(* Logix 5000 project; controller Ceca_1650T_Press 5069-L306ERM rev 32.11; software revision 32.02 *)

TASK MainTask (continuous, watchdog 500 ms) : MainProgram

MODULES
   Local : 5069-L306ERM (5069 0, rev 32.11)
      INPUT2 : vendor 1 type 7 code 1212 (5069 2, rev 3.1, StandardDataDriven RPI 5 ms)
      INPUT3 : vendor 1 type 7 code 1212 (5069 3, rev 3.1, StandardDataDriven RPI 5 ms)
      INPUT1 : vendor 1 type 7 code 1212 (5069 1, rev 3.1, StandardDataDriven RPI 5 ms)
      OUTPUT1 : vendor 1 type 7 code 1215 (5069 4, rev 3.1, StandardDataDriven RPI 5 ms)
      OUTPUT3 : vendor 1 type 7 code 1215 (5069 6, rev 3.1, StandardDataDriven RPI 5 ms)
      OUTPUT2 : vendor 1 type 7 code 1215 (5069 5, rev 3.1, StandardDataDriven RPI 5 ms)
END_MODULES

VAR_GLOBAL   (* controller tags *)
   AIR_SUPPLY_PRESSURE_DETECT : BOOL;
   AUTO_CYCLE_ENABLED : BOOL;   // M0014 HMI SELECTION
   AUTO_CYCLE_SELECTED : BOOL;   // HMI BUTTON/SELECTION B0102
   AUTO_CYCLE_STOP_PB : BOOL;
   AUTO_LOWER_LIMIT : BOOL;   // ENCODER SIGNAL B0155
   AUTO_ONE_CYCLE_ENABLED : BOOL;   // M0013 HMI SELECTION
   AUTO_ONE_CYCLE_SELECTED : BOOL;   // HMI BUTTON/SELECTION B0101
   AUTO_RESET_ALLOWED : BOOL;   // M003E
   AUTO_START_PB : BOOL;
   AUTO_START_PB_RESET : BOOL;
   AUTO_UPPER_LIMIT : BOOL;   // ENCODER SIGNAL B0151
   BLANKING_OFF_SIGNAL : TIMER := (PRE := 150);   // T0018
   BLANKING_PS_ENABLED : BOOL;   // M0018
   BOLSTER_CLAMP_OFF_LIMIT : BOOL;   // B0013
   BOLSTER_CLAMP_OFF_VALVE : BOOL;
   BOLSTER_CLAMP_ON : BOOL;   // M0006
   BOLSTER_CLAMP_ON_LIMIT : BOOL;   // B0012
   BOLSTER_CLAMP_ON_VALVE : BOOL;
   BOLSTER_DISABLED : BOOL;   // M0010
   BOLSTER_IN_ASSIST_LIMIT : BOOL;
   BOLSTER_IN_LIMIT : BOOL;   // B000E
   BOLSTER_IN_VALVE : BOOL;
   BOLSTER_LIFT_PRESSURE_DETECT : BOOL;
   BOLSTER_OUT_ASSIST_LIMIT : BOOL;
   BOLSTER_OUT_LIMIT : BOOL;
   BOLSTER_OUT_VALVE : BOOL;
   BOLSTER_REDUCTION_VALVE : BOOL;
   BOLSTER_TOUCH_LIMIT_1 : BOOL;   // B0014
   BOLSTER_TOUCH_LIMIT_2 : BOOL;   // B0015
   BOTH_DIE_CUSHIONS_DOWN : BOOL;   // M0036
   BUZZER_SIGNAL : BOOL;
   CANCEL_CYLINDER_LOWER_LIMIT : BOOL;
   CANCEL_DECOMPRESSION_VALVE : BOOL;
   CANCEL_HIGH_PRESSURE_VAVLE : BOOL;
   CANCEL_LOW_PRESSURE_VALVE : BOOL;
   CANCEL_UP_VALVE : BOOL;
   COOLING_WATER_ON_VALVE : BOOL;
   DC_POWER_ASSIST_VALVE : BOOL;
   DEBOUNCE_TIMER_LOCKING_OFF : TIMER := (PRE := 100);
   DEBOUNCE_TIMER_LOCKING_OFF_COMPLETE : TIMER := (PRE := 100);
   DECOMPRESSION : BOOL;   // M006D
   DIE_CHANGE_ENABLED : BOOL;   // M0015
   DIE_CHANGE_MODE : BOOL;   // HMI BUTTON/SELECTION B0103
   DIE_CUSHION_PB_OFF_STATE : BOOL;   // M003F
   DIE_DRAWRIC_CYLINDER_UPPER_PS : BOOL;   // B0018
   DIE_DRAWRIC_DECOMPRESSION_VALVE : BOOL;
   DIE_DRAWRIC_POWER_ASSIST_VALVE : BOOL;
   DIE_SET_CHANGING : BOOL;
   DIECUSHION_PUMP_UNLOADING_VALVE_1 : BOOL;
   DIECUSHION_PUMP_UNLOADING_VALVE_2 : BOOL;
   DIECUSHION_UPPER_LIMIT : BOOL;
   DRAW_ASSIST_COMPLETE : BOOL;   // M007D
   DRAW_BLANKING_NOT_SELECT : BOOL;   // M0017
   DRAW_UP_ASSIST : BOOL;   // M007C
   DRAWING_LS_ENABLED : BOOL;   // M0016????REMOVE????
   EMERGENCY_STOP : BOOL;
   ENABLE_1000T : BOOL;   // HMI BUTTON/RECIPE
   ENABLE_1500T : BOOL;   // HMI BUTTON/RECIPE
   ENABLE_500T : BOOL;   // HMI BUTTON/RECIPE
   FILTER_CHOKER : BOOL;
   FRONT_SHUTTER_SAFETY : BOOL;   // M002A
   FRONT_SUTTER_ON_LIMIT : BOOL;
   HALF_FINISHED_CYLINDER_ADVANCE_LIMIT : BOOL;
   HALF_FINISHED_CYLINDER_RETURN_LIMIT : BOOL;
   HALF_FINISHED_SUPPLY_VALVE : BOOL;
   INCH_ENABLED : BOOL;   // M0012 HMI SELECTION
   INCHING_SELECTED : BOOL;   // HMI BUTTON/SELECTION B0100
   L_DIECUSHION_AUTO_UP_LIMIT : BOOL;   // B0156 ENCODER SIGNAL
   L_DIECUSHION_DOWN : BOOL;   // M0003
   L_DIECUSHION_UP : BOOL;   // M0002
   LEFT_DIECUSHION_DECOMPRESSION_VALVE : BOOL;
   LEFT_DIECUSHION_DOWN_VALVE : BOOL;
   LEFT_DIECUSHION_LOWER_LIMIT : BOOL;   // B0006
   LEFT_DIECUSHION_POWER_ASSIST_VALVE : BOOL;
   LEFT_DIECUSHION_UP_VALVE : BOOL;
   LEFT_DIECUSHION_UPPER_LIMIT : BOOL;   // B0005
   LIFT_CYLINDER_DOWN_VALVE : BOOL;
   LIFT_CYLINDER_UP_VALVE : BOOL;
   LOCKING_OFF : BOOL;   // M0004
   LOCKING_OFF_ASSIST : BOOL;   // M0032
   LOCKING_OFF_COMPLETE : BOOL;   // M0033
   LOCKING_OFF_LIMIT : BOOL;   // B0007
   LOCKING_OFF_MEMORY : BOOL;   // M0031
   LOCKING_OFF_VALVE : BOOL;   // B0058
   LOCKING_ON : BOOL;   // M0005
   LOCKING_ON_LIMIT : BOOL;   // B0008
   LUBRICATION_OIL_LEVEL_DETECT : BOOL;
   LUBRICATION_PRESSURE_DETECT : BOOL;
   M_PRESS_DOWN : BOOL;   // M006A
   M_PRESS_DOWN_COMPLETE : BOOL;   // M006C
   M_PRESS_DOWN_COMPLETE_TIMER : TIMER := (PRE := 30);   // T0012
   M_PRESS_UP : BOOL;   // M006E
   M_PRESS_UP_COMPLETE : BOOL;   // M006F
   MAIN_DOWN_VALVE : BOOL;   // B0041
   MAIN_DOWN_VALVE_1000_TON : BOOL;   // B0043
   MAIN_DOWN_VALVE_500_TON : BOOL;   // B0042
   MAIN_LOWER_ASSIST_LIMIT : BOOL;   // B0026
   MAIN_LOWER_LIMIT : BOOL;   // B0002
   MAIN_NO_LOAD_VALVE : BOOL;   // B0046
   MAIN_POWER_HOLDING_VALVE : BOOL;   // B0045
   MAIN_PRESS_CONDITION_DOWN : BOOL;   // M0039
   MAIN_PRESS_CONDITION_UP : BOOL;   // M0038
   MAIN_PRESS_DOWN : BOOL;   // M0045
   MAIN_PRESS_DOWN_ASSIST : BOOL;   // M0044
   MAIN_PRESS_DOWN_MEMORY : BOOL;   // M006A
   MAIN_PRESS_NO_PRESSURE_DOWN : BOOL;   // M0047
   MAIN_PRESS_PRESSURE_DETECT : BOOL;   // B0016
   MAIN_PRESS_SLOW_DOWN : BOOL;   // M0046
   MAIN_PRESS_SLOW_DOWN_SIGNAL : BOOL;   // M0030
   MAIN_PRESS_SLOW_UP : BOOL;   // M0042
   MAIN_PRESS_UP : BOOL;   // M0041
   MAIN_PRESS_UP_ASSIST : BOOL;   // M0040
   MAIN_SLOW_DOWN_VALVE : BOOL;   // B0044
   MAIN_UP_VALVE : BOOL;   // B0040
   MAIN_UPPER_ASSIST : BOOL;   // B0001
   MAIN_UPPER_LIMIT : BOOL;   // B0000
   MOTOR_OVER_LOAD : BOOL;
   NO_PRESSUE_DOWN_PB : BOOL;   // B010D HMI BUTTON
   OIL_COOLER_START : BOOL;
   OIL_TEMP_TOO_HIGH : BOOL;
   OIL_TEMP_WARM_UP_START : BOOL;
   OPERATION_ON : BOOL;   // B0020
   PILOT_CHECK_OPEN_VALVE : BOOL;   // B0048
   PILOT_PUMP_HIGH_PRESSURE_VALVE : BOOL;
   PILOT_PUMP_MIDDLE_PRESSURE_VALVE : BOOL;
   PILOT_PUMP_ON : BOOL;
   PREFILL_VALVE_OPEN_VALVE : BOOL;   // B0047
   PREFILL_VALVE_OPEN_VALVE_2 : BOOL;
   PRESS_AUTO_CYCLE_SELECT_CONDITION : BOOL;   // M0060
   PRESS_AUTO_RUN : BOOL;   // M0069
   PRESS_HAS_A_FAULT_2 : BOOL;   // M0028
   PRESS_HOLDING_TIME : BOOL;   // M006B
   PRESS_HOLDING_TIMER : TIMER;   // PRESS HOLDING TIMER
   PRESS_READY_CONFIRM : BOOL;   // M0043
   PUMP_RUN : BOOL;   // B0021
   PUMP_STOP_SIGNAL : BOOL;
   R_DIECUSHION_AUTO_UP_LIMIT : BOOL;   // B0158 ENCODER SIGNAL
   R_DIECUSHION_DOWN : BOOL;   // M0001
   R_DIECUSHION_UP : BOOL;   // M0000
   REAR_SHUTTER_ON_LIMIT : BOOL;
   RIGHT_DIECUSHION_DECOMPRESSION_VALVE : BOOL;
   RIGHT_DIECUSHION_DOWN_VALVE : BOOL;
   RIGHT_DIECUSHION_LOWER_LIMIT : BOOL;   // B0004
   RIGHT_DIECUSHION_POWER_ASSIST_VALVE : BOOL;
   RIGHT_DIECUSHION_UP_VALVE : BOOL;
   RIGHT_DIECUSHION_UPPER_LIMIT : BOOL;   // B0003
   SAFETY_BAR_OPENED : BOOL;   // B000B
   SLIDE_DOWN_PB : BOOL;   // B010B HMI BUTTON
   SLIDE_SLOW_DOWN_PB : BOOL;   // B010C HMI BUTTON
   SLIDE_SLOW_DOWN_SIGNAL : BOOL;   // B0154 ENCODER SIGNAL
   SLIDE_SLOW_UP_PB : BOOL;   // B010A HMI BUTTON
   SLIDE_UP_PB : BOOL;   // HMI BUTTON B0109
   TIMER_OFF_DELAY_1500T : TIMER := (PRE := 50);   // T0017
   TIMER_OFF_DELAY_500T : TIMER := (PRE := 10);   // T0016
   UPPER_DIE_CLAMP_ON_DETECT : BOOL;
   UPPER_DIECLAMP_OFF_VALVE : BOOL;
   WARM_UP_OFF_TEMP : BOOL;
   WORK_LOCATION_VALVE : BOOL;
   WORKING_OIL_LEVEL_DETECT : BOOL;
END_VAR

PROGRAM MainProgram   (* main routine MainRoutine *)
VAR
   MESSAGES : STRING[100];
END_VAR

ROUTINE Bolster   (* ladder *)
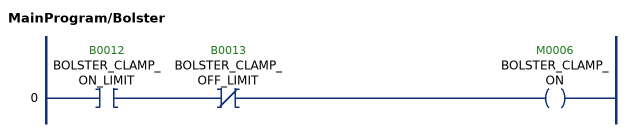
   0: XIC(BOLSTER_CLAMP_ON_LIMIT)XIO(BOLSTER_CLAMP_OFF_LIMIT)OTE(BOLSTER_CLAMP_ON);
END_ROUTINE

ROUTINE Cancel_Valves   (* ladder *)
END_ROUTINE

ROUTINE Die_Cushion   (* ladder *)
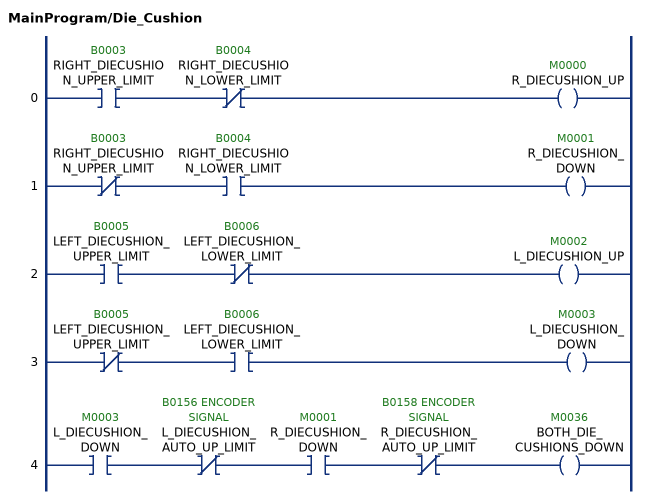
   0: XIC(RIGHT_DIECUSHION_UPPER_LIMIT)XIO(RIGHT_DIECUSHION_LOWER_LIMIT)OTE(R_DIECUSHION_UP);
   1: XIO(RIGHT_DIECUSHION_UPPER_LIMIT)XIC(RIGHT_DIECUSHION_LOWER_LIMIT)OTE(R_DIECUSHION_DOWN);
   2: XIC(LEFT_DIECUSHION_UPPER_LIMIT)XIO(LEFT_DIECUSHION_LOWER_LIMIT)OTE(L_DIECUSHION_UP);
   3: XIO(LEFT_DIECUSHION_UPPER_LIMIT)XIC(LEFT_DIECUSHION_LOWER_LIMIT)OTE(L_DIECUSHION_DOWN);
   4: XIC(L_DIECUSHION_DOWN)XIO(L_DIECUSHION_AUTO_UP_LIMIT)XIC(R_DIECUSHION_DOWN)XIO(R_DIECUSHION_AUTO_UP_LIMIT)OTE(BOTH_DIE_CUSHIONS_DOWN);
END_ROUTINE

ROUTINE Draw   (* ladder *)
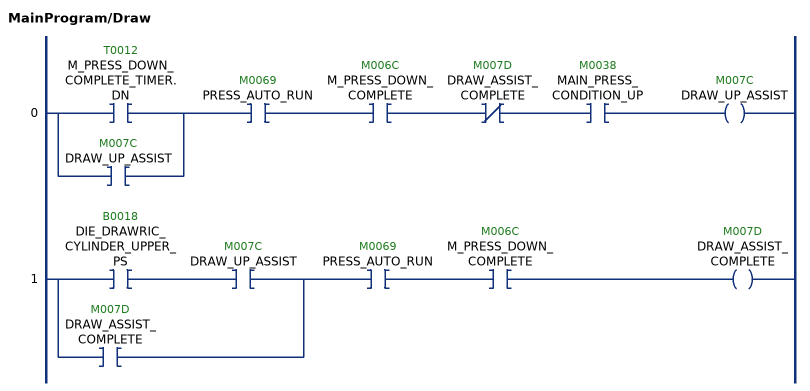
   0: [XIC(M_PRESS_DOWN_COMPLETE_TIMER.DN) ,XIC(DRAW_UP_ASSIST) ]XIC(PRESS_AUTO_RUN)XIC(M_PRESS_DOWN_COMPLETE)XIO(DRAW_ASSIST_COMPLETE)XIC(MAIN_PRESS_CONDITION_UP)OTE(DRAW_UP_ASSIST);
   1: [XIC(DIE_DRAWRIC_CYLINDER_UPPER_PS) XIC(DRAW_UP_ASSIST) ,XIC(DRAW_ASSIST_COMPLETE) ]XIC(PRESS_AUTO_RUN)XIC(M_PRESS_DOWN_COMPLETE)OTE(DRAW_ASSIST_COMPLETE);
END_ROUTINE

ROUTINE Inputs   (* ladder *)
   0: ;
END_ROUTINE

ROUTINE Locking   (* ladder *)
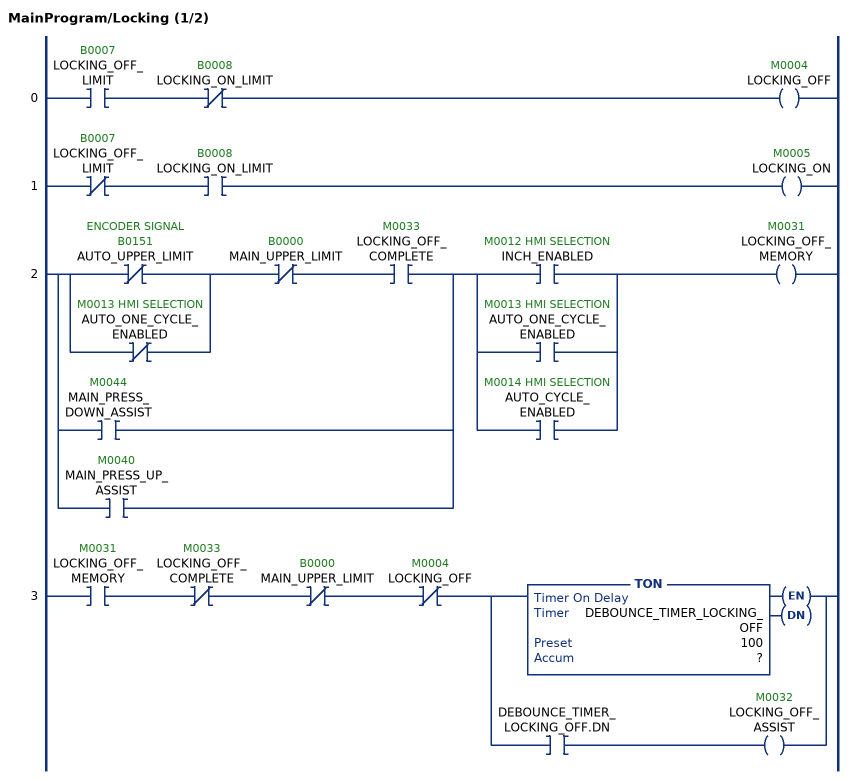
   0: XIC(LOCKING_OFF_LIMIT)XIO(LOCKING_ON_LIMIT)OTE(LOCKING_OFF);
   1: XIO(LOCKING_OFF_LIMIT)XIC(LOCKING_ON_LIMIT)OTE(LOCKING_ON);
   2: [[XIO(AUTO_UPPER_LIMIT) ,XIO(AUTO_ONE_CYCLE_ENABLED) ] XIO(MAIN_UPPER_LIMIT) XIC(LOCKING_OFF_COMPLETE) ,XIC(MAIN_PRESS_DOWN_ASSIST) ,XIC(MAIN_PRESS_UP_ASSIST) ][XIC(INCH_ENABLED) ,XIC(AUTO_ONE_CYCLE_ENABLED) ,XIC(AUTO_CYCLE_ENABLED) ]OTE(LOCKING_OFF_MEMORY);
   3: XIC(LOCKING_OFF_MEMORY)XIO(LOCKING_OFF_COMPLETE)XIO(MAIN_UPPER_LIMIT)XIO(LOCKING_OFF)[TON(DEBOUNCE_TIMER_LOCKING_OFF,?,?) ,XIC(DEBOUNCE_TIMER_LOCKING_OFF.DN) OTE(LOCKING_OFF_ASSIST) ];
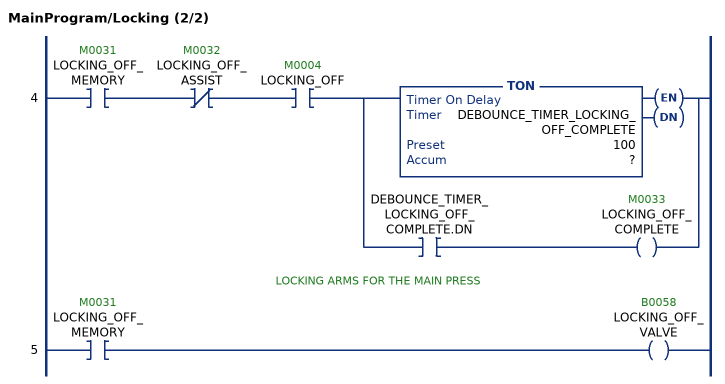
   4: XIC(LOCKING_OFF_MEMORY)XIO(LOCKING_OFF_ASSIST)XIC(LOCKING_OFF)[TON(DEBOUNCE_TIMER_LOCKING_OFF_COMPLETE,?,?) ,XIC(DEBOUNCE_TIMER_LOCKING_OFF_COMPLETE.DN) OTE(LOCKING_OFF_COMPLETE) ];
   // LOCKING ARMS FOR THE MAIN PRESS
   5: XIC(LOCKING_OFF_MEMORY)OTE(LOCKING_OFF_VALVE);
END_ROUTINE

ROUTINE Main_Down   (* ladder *)
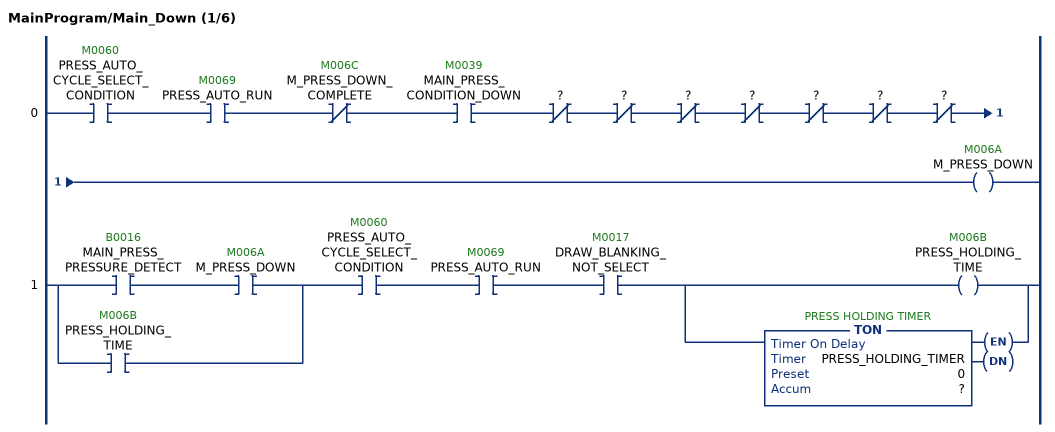
   0: XIC(PRESS_AUTO_CYCLE_SELECT_CONDITION)XIC(PRESS_AUTO_RUN)XIO(M_PRESS_DOWN_COMPLETE)XIC(MAIN_PRESS_CONDITION_DOWN)XIO(?)XIO(?)XIO(?)XIO(?)XIO(?)XIO(?)XIO(?)OTE(M_PRESS_DOWN);
   1: [XIC(MAIN_PRESS_PRESSURE_DETECT) XIC(M_PRESS_DOWN) ,XIC(PRESS_HOLDING_TIME) ]XIC(PRESS_AUTO_CYCLE_SELECT_CONDITION)XIC(PRESS_AUTO_RUN)XIC(DRAW_BLANKING_NOT_SELECT)[OTE(PRESS_HOLDING_TIME) ,TON(PRESS_HOLDING_TIMER,?,?) ];
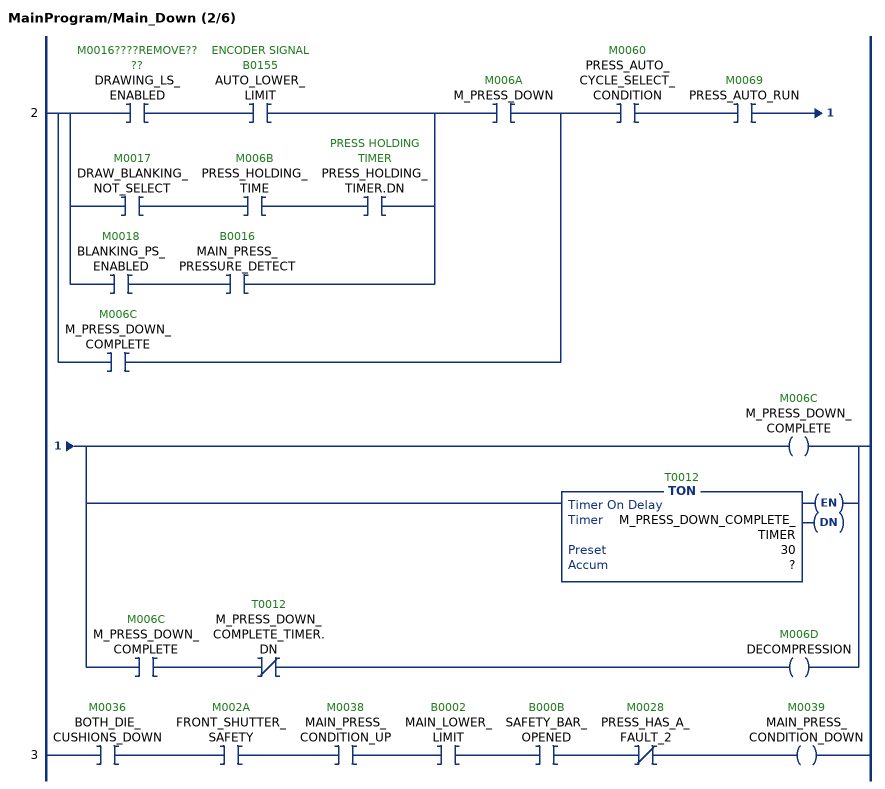
   2: [[XIC(DRAWING_LS_ENABLED) XIC(AUTO_LOWER_LIMIT) ,XIC(DRAW_BLANKING_NOT_SELECT) XIC(PRESS_HOLDING_TIME) XIC(PRESS_HOLDING_TIMER.DN) ,XIC(BLANKING_PS_ENABLED) XIC(MAIN_PRESS_PRESSURE_DETECT) ] XIC(M_PRESS_DOWN) ,XIC(M_PRESS_DOWN_COMPLETE) ]XIC(PRESS_AUTO_CYCLE_SELECT_CONDITION)XIC(PRESS_AUTO_RUN)[OTE(M_PRESS_DOWN_COMPLETE) ,TON(M_PRESS_DOWN_COMPLETE_TIMER,?,?) ,XIC(M_PRESS_DOWN_COMPLETE) XIO(M_PRESS_DOWN_COMPLETE_TIMER.DN) OTE(DECOMPRESSION) ];
   3: XIC(BOTH_DIE_CUSHIONS_DOWN)XIC(FRONT_SHUTTER_SAFETY)XIC(MAIN_PRESS_CONDITION_UP)XIC(MAIN_LOWER_LIMIT)XIC(SAFETY_BAR_OPENED)XIO(PRESS_HAS_A_FAULT_2)OTE(MAIN_PRESS_CONDITION_DOWN);
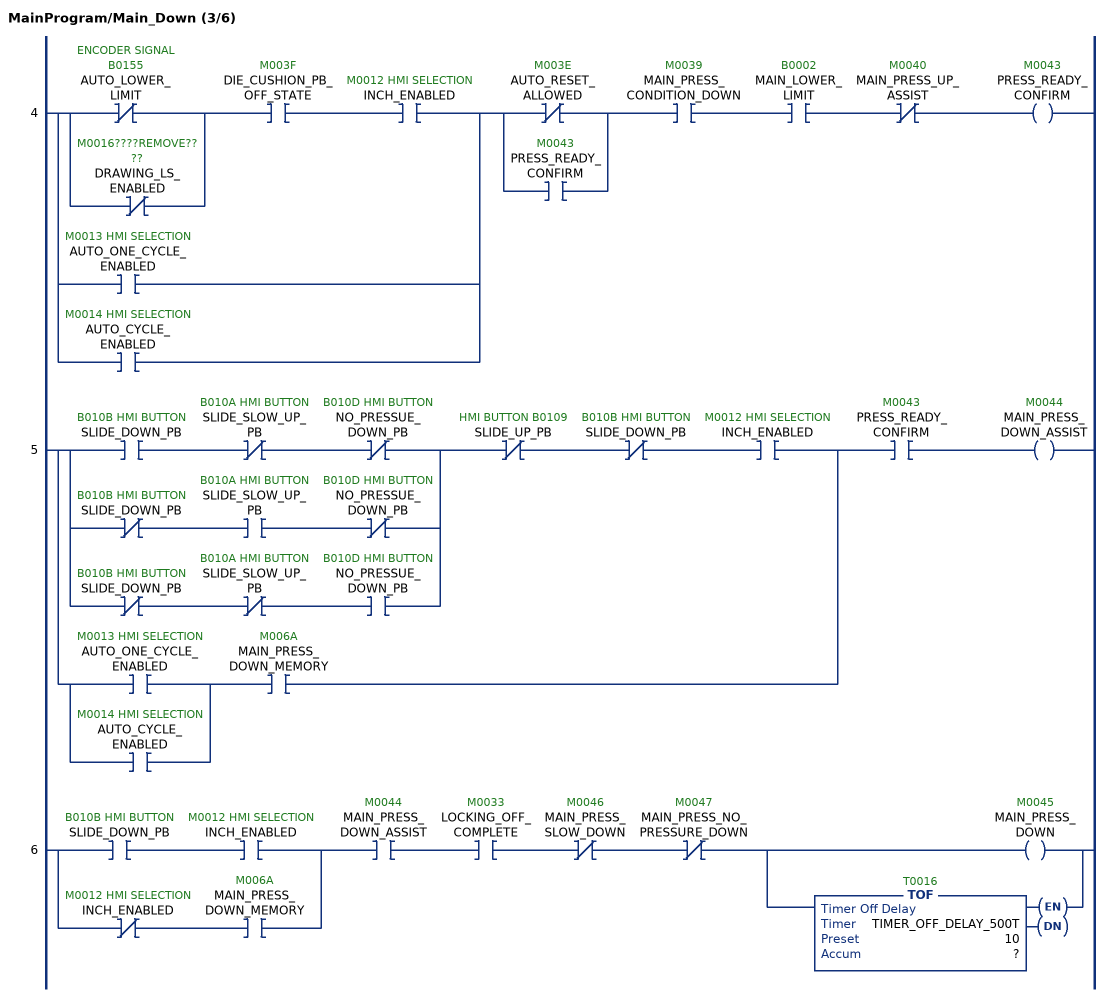
   4: [[XIO(AUTO_LOWER_LIMIT) ,XIO(DRAWING_LS_ENABLED) ] XIC(DIE_CUSHION_PB_OFF_STATE) XIC(INCH_ENABLED) ,XIC(AUTO_ONE_CYCLE_ENABLED) ,XIC(AUTO_CYCLE_ENABLED) ][XIO(AUTO_RESET_ALLOWED) ,XIC(PRESS_READY_CONFIRM) ]XIC(MAIN_PRESS_CONDITION_DOWN)XIC(MAIN_LOWER_LIMIT)XIO(MAIN_PRESS_UP_ASSIST)OTE(PRESS_READY_CONFIRM);
   5: [[XIC(SLIDE_DOWN_PB) XIO(SLIDE_SLOW_UP_PB) XIO(NO_PRESSUE_DOWN_PB) ,XIO(SLIDE_DOWN_PB) XIC(SLIDE_SLOW_UP_PB) XIO(NO_PRESSUE_DOWN_PB) ,XIO(SLIDE_DOWN_PB) XIO(SLIDE_SLOW_UP_PB) XIC(NO_PRESSUE_DOWN_PB) ] XIO(SLIDE_UP_PB) XIO(SLIDE_DOWN_PB) XIC(INCH_ENABLED) ,[XIC(AUTO_ONE_CYCLE_ENABLED) ,XIC(AUTO_CYCLE_ENABLED) ] XIC(MAIN_PRESS_DOWN_MEMORY) ]XIC(PRESS_READY_CONFIRM)OTE(MAIN_PRESS_DOWN_ASSIST);
   6: [XIC(SLIDE_DOWN_PB) XIC(INCH_ENABLED) ,XIO(INCH_ENABLED) XIC(MAIN_PRESS_DOWN_MEMORY) ]XIC(MAIN_PRESS_DOWN_ASSIST)XIC(LOCKING_OFF_COMPLETE)XIO(MAIN_PRESS_SLOW_DOWN)XIO(MAIN_PRESS_NO_PRESSURE_DOWN)[OTE(MAIN_PRESS_DOWN) ,TOF(TIMER_OFF_DELAY_500T,?,?) ];
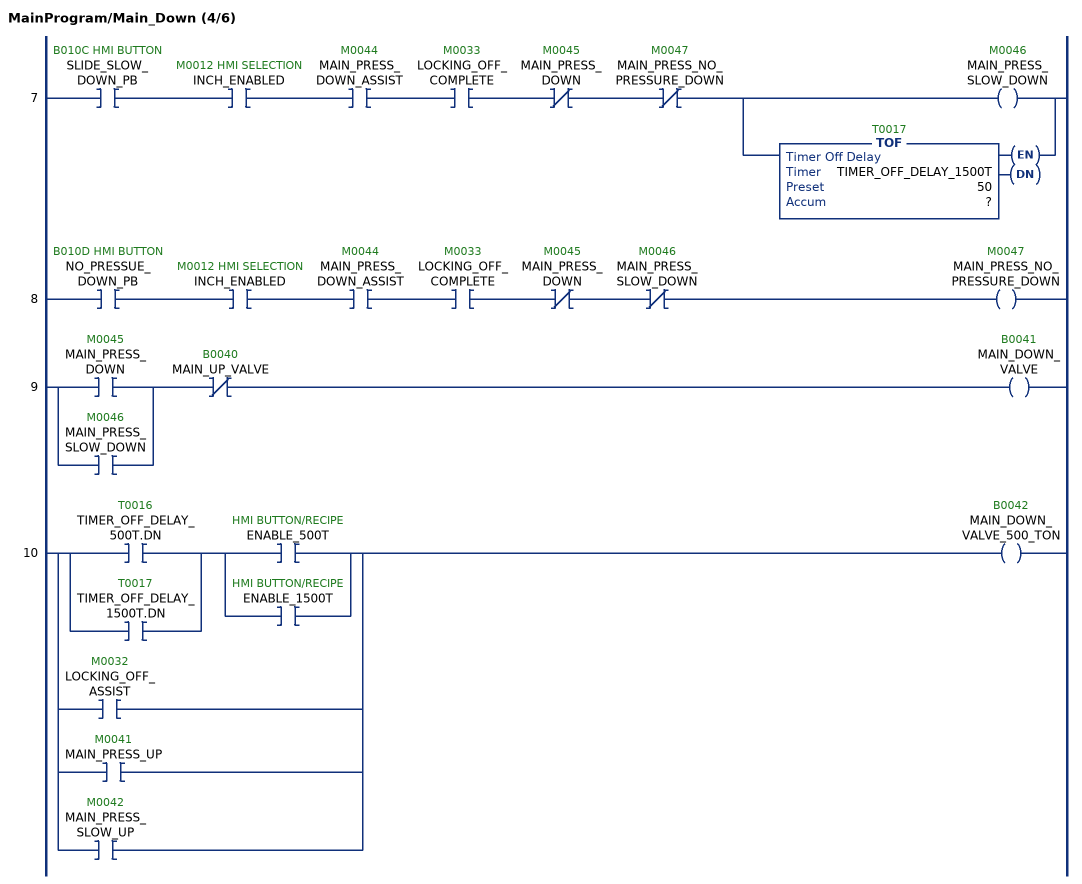
   7: XIC(SLIDE_SLOW_DOWN_PB)XIC(INCH_ENABLED)XIC(MAIN_PRESS_DOWN_ASSIST)XIC(LOCKING_OFF_COMPLETE)XIO(MAIN_PRESS_DOWN)XIO(MAIN_PRESS_NO_PRESSURE_DOWN)[OTE(MAIN_PRESS_SLOW_DOWN) ,TOF(TIMER_OFF_DELAY_1500T,?,?) ];
   8: XIC(NO_PRESSUE_DOWN_PB)XIC(INCH_ENABLED)XIC(MAIN_PRESS_DOWN_ASSIST)XIC(LOCKING_OFF_COMPLETE)XIO(MAIN_PRESS_DOWN)XIO(MAIN_PRESS_SLOW_DOWN)OTE(MAIN_PRESS_NO_PRESSURE_DOWN);
   9: [XIC(MAIN_PRESS_DOWN) ,XIC(MAIN_PRESS_SLOW_DOWN) ]XIO(MAIN_UP_VALVE)OTE(MAIN_DOWN_VALVE);
   10: [[XIC(TIMER_OFF_DELAY_500T.DN) ,XIC(TIMER_OFF_DELAY_1500T.DN) ] [XIC(ENABLE_500T) ,XIC(ENABLE_1500T) ] ,XIC(LOCKING_OFF_ASSIST) ,XIC(MAIN_PRESS_UP) ,XIC(MAIN_PRESS_SLOW_UP) ]OTE(MAIN_DOWN_VALVE_500_TON);
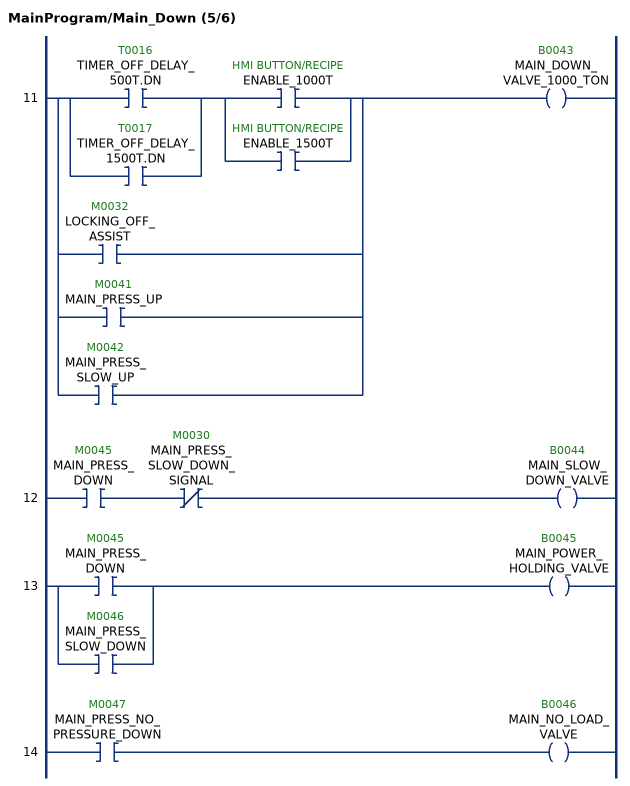
   11: [[XIC(TIMER_OFF_DELAY_500T.DN) ,XIC(TIMER_OFF_DELAY_1500T.DN) ] [XIC(ENABLE_1000T) ,XIC(ENABLE_1500T) ] ,XIC(LOCKING_OFF_ASSIST) ,XIC(MAIN_PRESS_UP) ,XIC(MAIN_PRESS_SLOW_UP) ]OTE(MAIN_DOWN_VALVE_1000_TON);
   12: XIC(MAIN_PRESS_DOWN)XIO(MAIN_PRESS_SLOW_DOWN_SIGNAL)OTE(MAIN_SLOW_DOWN_VALVE);
   13: [XIC(MAIN_PRESS_DOWN) ,XIC(MAIN_PRESS_SLOW_DOWN) ]OTE(MAIN_POWER_HOLDING_VALVE);
   14: XIC(MAIN_PRESS_NO_PRESSURE_DOWN)OTE(MAIN_NO_LOAD_VALVE);
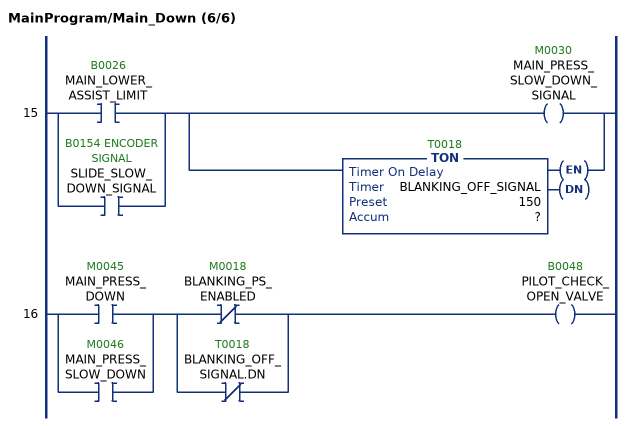
   15: [XIC(MAIN_LOWER_ASSIST_LIMIT) ,XIC(SLIDE_SLOW_DOWN_SIGNAL) ][OTE(MAIN_PRESS_SLOW_DOWN_SIGNAL) ,TON(BLANKING_OFF_SIGNAL,?,?) ];
   16: [XIC(MAIN_PRESS_DOWN) ,XIC(MAIN_PRESS_SLOW_DOWN) ][XIO(BLANKING_PS_ENABLED) ,XIO(BLANKING_OFF_SIGNAL.DN) ]OTE(PILOT_CHECK_OPEN_VALVE);
END_ROUTINE

ROUTINE Main_Up   (* ladder *)
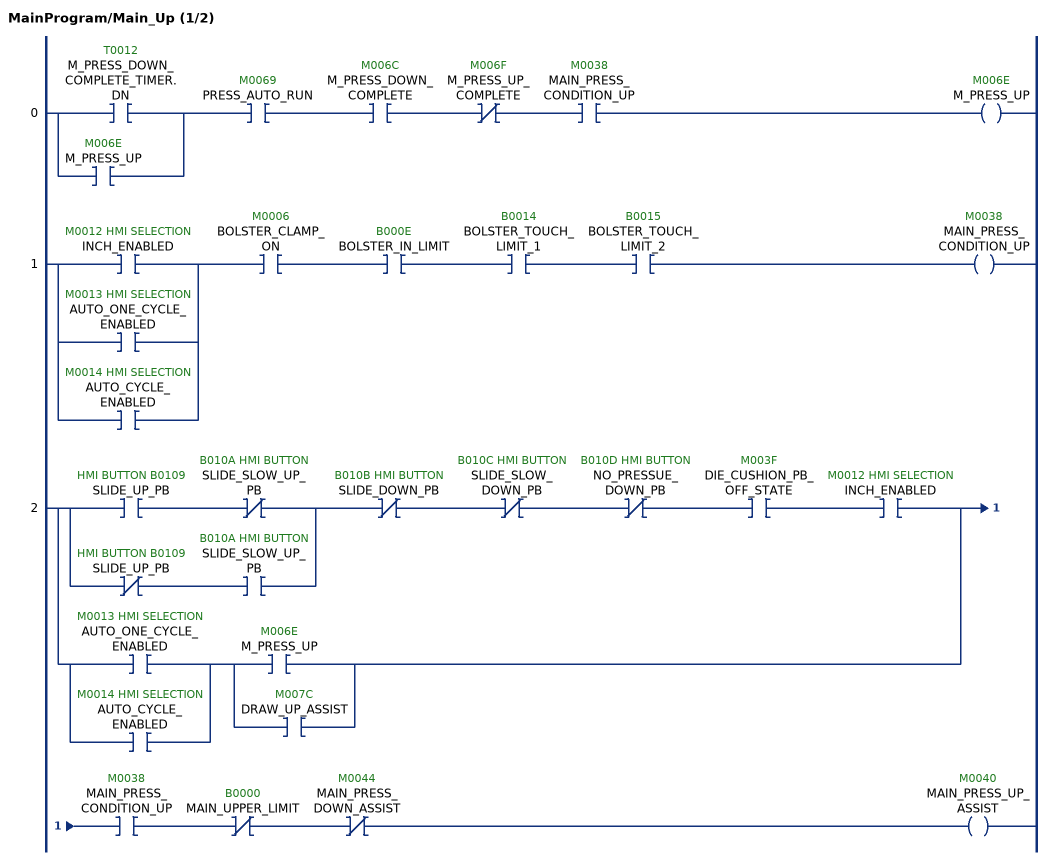
   0: [XIC(M_PRESS_DOWN_COMPLETE_TIMER.DN) ,XIC(M_PRESS_UP) ]XIC(PRESS_AUTO_RUN)XIC(M_PRESS_DOWN_COMPLETE)XIO(M_PRESS_UP_COMPLETE)XIC(MAIN_PRESS_CONDITION_UP)OTE(M_PRESS_UP);
   1: [XIC(INCH_ENABLED) ,XIC(AUTO_ONE_CYCLE_ENABLED) ,XIC(AUTO_CYCLE_ENABLED) ]XIC(BOLSTER_CLAMP_ON)XIC(BOLSTER_IN_LIMIT)XIC(BOLSTER_TOUCH_LIMIT_1)XIC(BOLSTER_TOUCH_LIMIT_2)OTE(MAIN_PRESS_CONDITION_UP);
   2: [[XIC(SLIDE_UP_PB) XIO(SLIDE_SLOW_UP_PB) ,XIO(SLIDE_UP_PB) XIC(SLIDE_SLOW_UP_PB) ] XIO(SLIDE_DOWN_PB) XIO(SLIDE_SLOW_DOWN_PB) XIO(NO_PRESSUE_DOWN_PB) XIC(DIE_CUSHION_PB_OFF_STATE) XIC(INCH_ENABLED) ,[XIC(AUTO_ONE_CYCLE_ENABLED) ,XIC(AUTO_CYCLE_ENABLED) ] [XIC(M_PRESS_UP) ,XIC(DRAW_UP_ASSIST) ] ]XIC(MAIN_PRESS_CONDITION_UP)XIO(MAIN_UPPER_LIMIT)XIO(MAIN_PRESS_DOWN_ASSIST)OTE(MAIN_PRESS_UP_ASSIST);
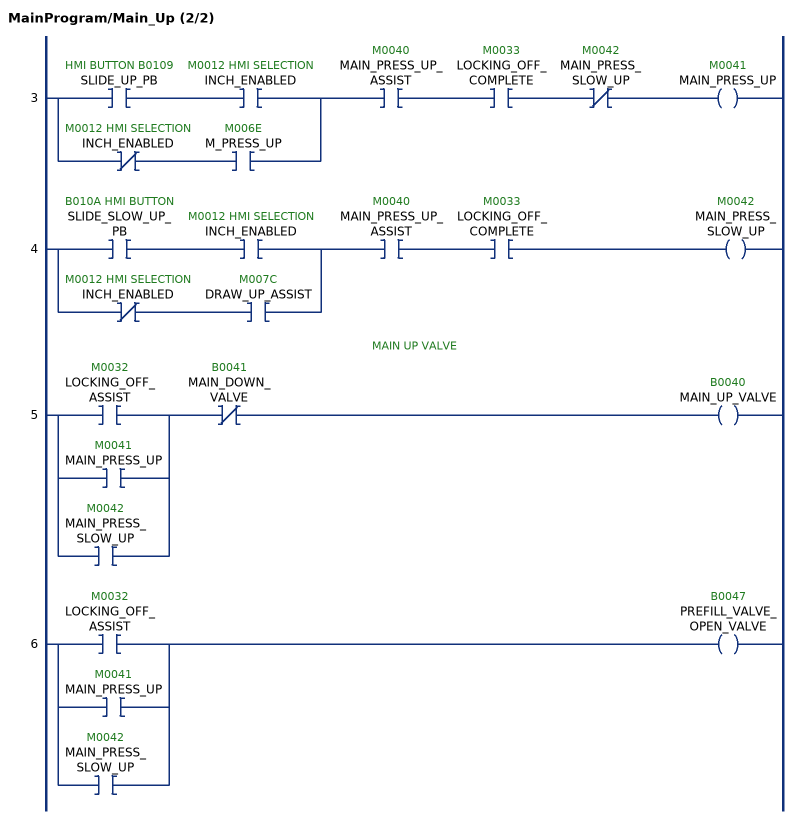
   3: [XIC(SLIDE_UP_PB) XIC(INCH_ENABLED) ,XIO(INCH_ENABLED) XIC(M_PRESS_UP) ]XIC(MAIN_PRESS_UP_ASSIST)XIC(LOCKING_OFF_COMPLETE)XIO(MAIN_PRESS_SLOW_UP)OTE(MAIN_PRESS_UP);
   4: [XIC(SLIDE_SLOW_UP_PB) XIC(INCH_ENABLED) ,XIO(INCH_ENABLED) XIC(DRAW_UP_ASSIST) ]XIC(MAIN_PRESS_UP_ASSIST)XIC(LOCKING_OFF_COMPLETE)OTE(MAIN_PRESS_SLOW_UP);
   // MAIN UP VALVE
   5: [XIC(LOCKING_OFF_ASSIST) ,XIC(MAIN_PRESS_UP) ,XIC(MAIN_PRESS_SLOW_UP) ]XIO(MAIN_DOWN_VALVE)OTE(MAIN_UP_VALVE);
   6: [XIC(LOCKING_OFF_ASSIST) ,XIC(MAIN_PRESS_UP) ,XIC(MAIN_PRESS_SLOW_UP) ]OTE(PREFILL_VALVE_OPEN_VALVE);
END_ROUTINE

ROUTINE MainRoutine   (* ladder *)
END_ROUTINE

ROUTINE Messages   (* ladder *)
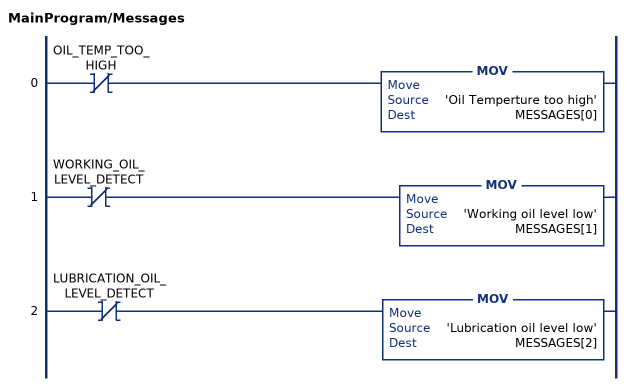
   0: XIO(OIL_TEMP_TOO_HIGH)MOV('Oil Temperture too high',MESSAGES[0]);
   1: XIO(WORKING_OIL_LEVEL_DETECT)MOV('Working oil level low',MESSAGES[1]);
   2: XIO(LUBRICATION_OIL_LEVEL_DETECT)MOV('Lubrication oil level low',MESSAGES[2]);
END_ROUTINE

ROUTINE Modes   (* ladder *)
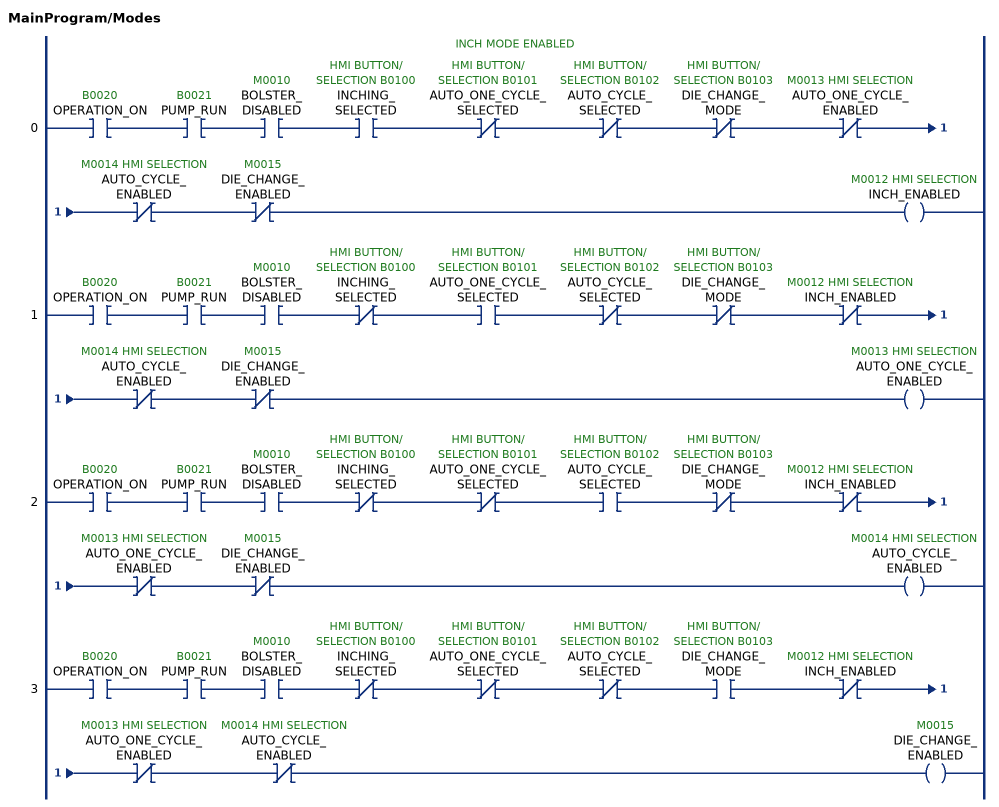
   // INCH MODE ENABLED
   0: XIC(OPERATION_ON)XIC(PUMP_RUN)XIC(BOLSTER_DISABLED)XIC(INCHING_SELECTED)XIO(AUTO_ONE_CYCLE_SELECTED)XIO(AUTO_CYCLE_SELECTED)XIO(DIE_CHANGE_MODE)XIO(AUTO_ONE_CYCLE_ENABLED)XIO(AUTO_CYCLE_ENABLED)XIO(DIE_CHANGE_ENABLED)OTE(INCH_ENABLED);
   1: XIC(OPERATION_ON)XIC(PUMP_RUN)XIC(BOLSTER_DISABLED)XIO(INCHING_SELECTED)XIC(AUTO_ONE_CYCLE_SELECTED)XIO(AUTO_CYCLE_SELECTED)XIO(DIE_CHANGE_MODE)XIO(INCH_ENABLED)XIO(AUTO_CYCLE_ENABLED)XIO(DIE_CHANGE_ENABLED)OTE(AUTO_ONE_CYCLE_ENABLED);
   2: XIC(OPERATION_ON)XIC(PUMP_RUN)XIC(BOLSTER_DISABLED)XIO(INCHING_SELECTED)XIO(AUTO_ONE_CYCLE_SELECTED)XIC(AUTO_CYCLE_SELECTED)XIO(DIE_CHANGE_MODE)XIO(INCH_ENABLED)XIO(AUTO_ONE_CYCLE_ENABLED)XIO(DIE_CHANGE_ENABLED)OTE(AUTO_CYCLE_ENABLED);
   3: XIC(OPERATION_ON)XIC(PUMP_RUN)XIC(BOLSTER_DISABLED)XIO(INCHING_SELECTED)XIO(AUTO_ONE_CYCLE_SELECTED)XIO(AUTO_CYCLE_SELECTED)XIC(DIE_CHANGE_MODE)XIO(INCH_ENABLED)XIO(AUTO_ONE_CYCLE_ENABLED)XIO(AUTO_CYCLE_ENABLED)OTE(DIE_CHANGE_ENABLED);
END_ROUTINE

ROUTINE Outputs   (* ladder *)
   0: ;
END_ROUTINE

ROUTINE Safety   (* ladder *)
   0: ;
END_ROUTINE

ROUTINE Valves   (* ladder *)
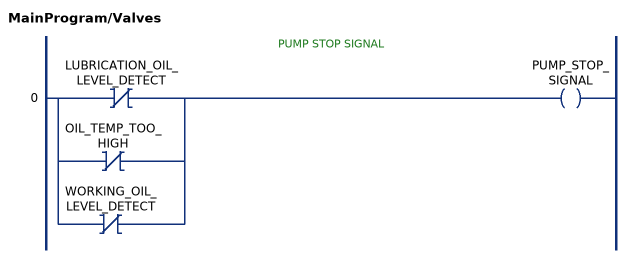
   // PUMP STOP SIGNAL
   0: [XIO(LUBRICATION_OIL_LEVEL_DETECT) ,XIO(OIL_TEMP_TOO_HIGH) ,XIO(WORKING_OIL_LEVEL_DETECT) ]OTE(PUMP_STOP_SIGNAL);
END_ROUTINE
END_PROGRAM
